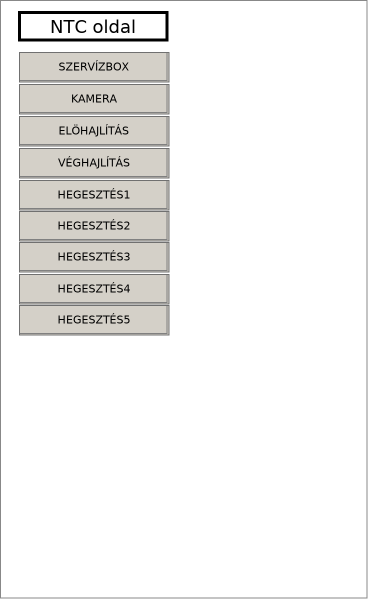
VISUALIZATION Tengely_NTC_beallitasok  // 368x599
    Label (297,567 69x30)
    RoundedRectangle (18,11 150x30)
    Label (18,12 150x30), "NTC oldal"
    Button (19,116 150x30), "ELÖHAJLÍTÁS"
        OnMouseUp: execute { GVL.iFoLapozo:=GVL.SZERVIZ_FUL; GVL.iSzervizLapozo:=GVL.HAJLITOK_FUL; }
    Button (19,148 150x30), "VÉGHAJLÍTÁS"
        OnMouseUp: execute { GVL.iFoLapozo:=GVL.SZERVIZ_FUL; GVL.iSzervizLapozo:=GVL.HAJLITOK_FUL; }
    Button (19,180 150x30), "HEGESZTÉS1"
        OnMouseUp: execute {
            GVL.iFoLapozo:=GVL.SZERVIZ_FUL;
            GVL.iSzervizLapozo:=GVL.HEGESZTES_FUL;
            GVL.iTengelyLapozo:=GVL.NTC_TENGELY_FUL;
        }
    Button (19,211 150x30), "HEGESZTÉS2"
        OnMouseUp: execute {
            GVL.iFoLapozo:=GVL.SZERVIZ_FUL;
            GVL.iSzervizLapozo:=GVL.HEGESZTES_FUL;
            GVL.iTengelyLapozo:=GVL.NTC_TENGELY_FUL;
        }
    Button (19,242 150x30), "HEGESZTÉS3"
        OnMouseUp: execute {
            GVL.iFoLapozo:=GVL.SZERVIZ_FUL;
            GVL.iSzervizLapozo:=GVL.HEGESZTES_FUL;
            GVL.iTengelyLapozo:=GVL.NTC_TENGELY_FUL;
        }
    Button (19,274 150x30), "HEGESZTÉS4"
        OnMouseUp: execute {
            GVL.iFoLapozo:=GVL.SZERVIZ_FUL;
            GVL.iSzervizLapozo:=GVL.HEGESZTES_FUL;
            GVL.iTengelyLapozo:=GVL.NTC_TENGELY_FUL;
        }
    Button (19,305 150x30), "HEGESZTÉS5"
        OnMouseUp: execute {
            GVL.iFoLapozo:=GVL.SZERVIZ_FUL;
            GVL.iSzervizLapozo:=GVL.HEGESZTES_FUL;
            GVL.iTengelyLapozo:=GVL.NTC_TENGELY_FUL;
        }
    Button (19,52 150x30), "SZERVÍZBOX"
        OnMouseUp: execute { GVL.iFoLapozo:=GVL.SZERVIZ_FUL; GVL.iSzervizLapozo:=GVL.BEHELYEZES_FUL; }
    Button (19,84 150x30), "KAMERA"
        OnMouseUp: execute { GVL.iFoLapozo:=GVL.SZERVIZ_FUL; GVL.iSzervizLapozo:=GVL.BEHELYEZES_FUL; }
END_VISUALIZATION

(* stored: Version 1.1.0.1, ProductVersion 3.1.4024.11
   Visu Tengely_NTC_beallitasok: Id {9d0f6fb3-8233-4b6c-9f2d-4b9c252554da} *)
